TYPE MotorI :
STRUCT
	Start : BOOL;
	Stop : BOOL;
	Overload : BOOL;
	ResetOverload: BOOL;
END_STRUCT
END_TYPE

(* stored: Version 1.1.0.1, ProductVersion 3.1.4024.12
   DUT MotorI: Id {9ab7ac65-9eff-405d-af25-e0d1d99f28e5} *)
